// Returns current task cycle time in seconds.
FUNCTION GetTaskCycleTime : LREAL
VAR_IN_OUT CONSTANT
	taskInfo: ARRAY[*] OF PlcTaskSystemInfo; // Pass application _TaskInfo.
END_VAR

GetTaskCycleTime := UDINT_TO_LREAL(taskInfo[TC2_System.GETCURTASKINDEXEX()].CycleTime) / 10_000_000;

END_FUNCTION

(* stored: Version 1.1.0.1
   POU GetTaskCycleTime: Id {da69abd6-8927-4295-ac94-a73a8afb23e1}, SpecialFunc None *)
